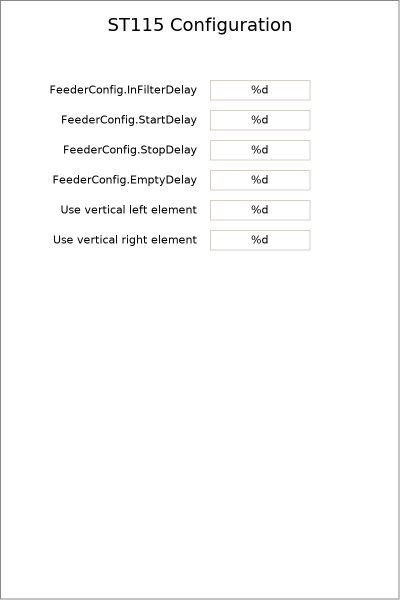
VISUALIZATION VISU_Recipe_ST115  // 400x600
    Textfield (210,80 100x20), "%d", text variable: _20_AUTO.recipe.st115.FeederConfig.InFilterDelay
        OnMouseDown: write the text variable via Default
    Label (0,5 400x40), "ST115 Configuration"
    Label (0,80 200x20), "FeederConfig.InFilterDelay"
    Textfield (210,110 100x20), "%d", text variable: _20_AUTO.recipe.st115.FeederConfig.StartDelay
        OnMouseDown: write the text variable via Default
    Label (0,110 200x20), "FeederConfig.StartDelay"
    Textfield (210,140 100x20), "%d", text variable: _20_AUTO.recipe.st115.FeederConfig.StopDelay
        OnMouseDown: write the text variable via Default
    Label (0,140 200x20), "FeederConfig.StopDelay"
    Textfield (210,170 100x20), "%d", text variable: _20_AUTO.recipe.st115.FeederConfig.EmptyDelay
        OnMouseDown: write the text variable via Default
    Label (0,170 200x20), "FeederConfig.EmptyDelay"
    Label (0,200 200x20), "Use vertical left element"
    Label (0,230 200x20), "Use vertical right element"
    Textfield (210,200 100x20), "%d", text variable: _20_AUTO.recipe.st115.xUseVerLeft
        OnMouseDown: write the text variable via Default
    Textfield (210,230 100x20), "%d", text variable: _20_AUTO.recipe.st115.xUseVerRight
        OnMouseDown: write the text variable via Default
END_VISUALIZATION

(* stored: Version 1.1.0.1, ProductVersion 3.1.4024.6
   Visu VISU_Recipe_ST115: Id {2c9824aa-7864-4a05-a566-e5bb98a0fbab} *)
